# EPICS StreamDevice protocol: siteApps/IF-Motor-Control-1-0/proto/ls224.proto
terminator = CR LF;

replytimeout = 3000;
readtimeout = 1000;

read_kelvin {out "KRDG? \$1"; in "%f";}
reset {out "*RST";}
